// TIA Portal project "Project2" (V17)

(* hardware
DEVICE "S7-1200 station_1"  S7-1200 Station
   slot 0: "Rack_0"  S7-1200 Rack  Rack  V1.0
   slot 1: "PLC_1"  CPU 1214C AC/DC/Rly  6ES7 214-1BG40-0XB0  V4.2
*)

// ===== PLC "PLC_1"  CPU 1214C AC/DC/Rly =====

VAR_GLOBAL   // PLC tag table "Default tag table"
   "IN00" AT %I0.0 : Bool;
   "IN01" AT %I0.1 : Bool;
   "IN02" AT %I0.2 : Bool;
   "IN03" AT %I0.3 : Bool;
   "OUT00" AT %Q0.0 : Bool;
   "OUT01" AT %Q0.1 : Bool;
   "OUT02" AT %Q0.2 : Bool;
   "OUT03" AT %Q0.3 : Bool;
   "OUT04" AT %Q0.4 : Bool;
   "OUT05" AT %Q0.5 : Bool;
END_VAR

ORGANIZATION_BLOCK "Main"   // OB1, LAD, ProgramCycle
TITLE = "Main Program Sweep (Cycle)"
{ S7_Optimized_Access := 'TRUE' }
VERSION : 0.1
   VAR_INPUT
      Initial_Call : Bool;   // Initial call of this OB
      Remanence : Bool;   // =True, if remanent data are available
   END_VAR
BEGIN

REGION Network 1: AND
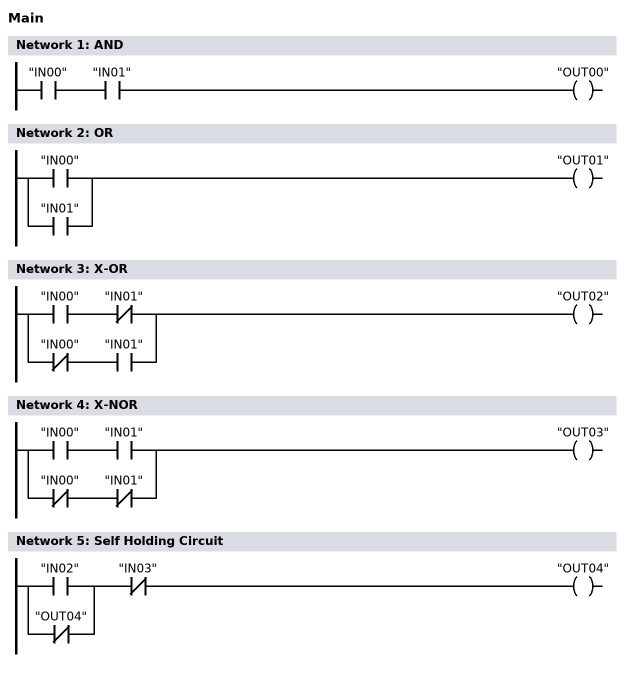
   RUNG wire#powerrail
      Contact( "IN00" )
      Contact( "IN01" )
      Coil( "OUT00" )
   END_RUNG
   // the same network as SCL:
   "OUT00" := "IN00" AND "IN01";
END_REGION

REGION Network 2: OR
   RUNG wire#powerrail
      Contact( "IN00" )
      wire#w1
      Coil( "OUT01" )
   END_RUNG
   RUNG wire#powerrail
      Contact( "IN01" )
   END_RUNG wire#w1
   // the same network as SCL:
   "OUT01" := "IN00" OR "IN01";
END_REGION

REGION Network 3: X-OR
   RUNG wire#powerrail
      Contact( "IN00" )
      I_Contact( "IN01" )
      wire#w1
      Coil( "OUT02" )
   END_RUNG
   RUNG wire#powerrail
      I_Contact( "IN00" )
      Contact( "IN01" )
   END_RUNG wire#w1
   // the same network as SCL:
   "OUT02" := ("IN00" AND NOT "IN01") OR (NOT "IN00" AND "IN01");
END_REGION

REGION Network 4: X-NOR
   RUNG wire#powerrail
      Contact( "IN00" )
      Contact( "IN01" )
      wire#w1
      Coil( "OUT03" )
   END_RUNG
   RUNG wire#powerrail
      I_Contact( "IN00" )
      I_Contact( "IN01" )
   END_RUNG wire#w1
   // the same network as SCL:
   "OUT03" := ("IN00" AND "IN01") OR (NOT "IN00" AND NOT "IN01");
END_REGION

REGION Network 5: Self Holding Circuit
   RUNG wire#powerrail
      Contact( "IN02" )
      wire#w1
      I_Contact( "IN03" )
      Coil( "OUT04" )
   END_RUNG
   RUNG wire#powerrail
      I_Contact( "OUT04" )
   END_RUNG wire#w1
   // the same network as SCL:
   "OUT04" := ("IN02" OR NOT "OUT04") AND NOT "IN03";
END_REGION
END_ORGANIZATION_BLOCK